(* PLC project  *)

CONFIGURATION XI110116
END_CONFIGURATION
